{attribute addProperty BoxType "KL2642-0050"}
{attribute addProperty Id "State_RelayAT %I*BOOL000OutputAT %Q*BOOL000"}
{attribute addProperty CRC "1022788430"}
{attribute addProperty SizeInBites "0"}
{attribute addProperty SizeInBytes "0"}
TYPE Channel_3CF6834E :
STRUCT
	{attribute addProperty Name "State_Relay"}
	State_Relay AT %I* : BOOL;
	{attribute addProperty Name "Output"}
	Output AT %Q* : BOOL;
END_STRUCT
END_TYPE

(* stored: Version 1.2.0.0, ProductVersion 3.1.4024.9
   DUT Channel_3CF6834E: Id {afd5c9a0-c3c4-4b8e-a3ba-1c1efbcc38d3} *)
